PROGRAM Prg_Counter
VAR
END_VAR

END_PROGRAM

(* stored: Version 1.1.0.1, ProductVersion 3.1.4024.9
   POU Prg_Counter: Id {56949bcf-47d4-4045-9858-74c2a0ec070a}, SpecialFunc None *)
